// TIA Portal V20 export
// export: Created 2025-12-01T14:56:22.0639924Z, ExportSetting None, DisplayName Totally Integrated Automation Portal, DisplayVersion V20 Update 3, DisplayName TIA Portal Openness, DisplayVersion V20 Update 3, DisplayName TIA Portal Version Control Interface, DisplayVersion V20 Update 3, DisplayName STEP 7 Professional, DisplayVersion V20 Update 3, DisplayName STEP 7 Safety, DisplayVersion V20 Update 2, DisplayName WinCC Basic/Comfort/Advanced, DisplayVersion V20 Update 3, DisplayName WinCC Professional, DisplayVersion V20 Update 3, DisplayName WinCC Unified, DisplayVersion V20 Update 3
TYPE "NDD_Interlock_Garras"
   STRUCT
      PosGarra_Bloqueo : Bool;
      MovGarra_Bloqueada : Bool;
      OrdenDeSalida : Bool;
      FinOrdenDeSalida : Bool;
      DejarCarga_EntradaGarra : Bool;
      DejadaCarga_EntradaGarra : Bool;
      RecogerCarga_SalidaGarra : Bool;
      RecogidaCarga_SalidaGarra : Bool;
      AVTF_EntradaGarra : Bool;   // Aviso de Entrada de la Paleta en la Garrauilla
      PTF_EntradaGarra : Bool;   // Permiso de Entrada de la Paleta en la Garrauilla
      FTF_EntradaGarra : Bool;   // Fin de la Entrada de la Paleta en la Garrauilla
      AVTF_SalidaGarra : Bool;   // Aviso de Salida de la Paleta en la Garrauilla
      PTF_SalidaGarra : Bool;   // Permiso de Salida de la Paleta en la Hoquilla
      FTF_SalidaGarra : Bool;   // Fin de la Salida de la Paleta en la Hoprquilla
      Libre_16 : Bool;
      DesHabilitarBarrera_Up : Bool;
      PuestoCarga_EnGarras : Bool;
      MA_Baliza_Garras : Bool;
      ConCarga_Garras : Bool;
      PosGarrasTransfer_OK : Bool;
      Garra_InicioPaletizado : Bool;
      Garra_FinPaletizado : Bool;
      Garra_Escondida : Bool;
      Garra_EnReset : Bool;
      Garra_EnCarga : Bool;
      Garra_EnVacio : Bool;
      Garra_Entrando { ExternalVisible := 'False'} : Bool;
      Garra_Saliendo : Bool;
      Libre_35 : Bool;
      Libre_36 : Bool;
      Libre_37 : Bool;
   END_STRUCT;
END_TYPE
